(* IEC 61131-3 sources: ATCMcontrol_Engineering/src/COM/softing/fc/AddOns/Softing/4CPCTarget/Libs/ATCM_IEC1131_3/table_37, 6 files *)

(* ---- tof.st ---- *)
(*[[
    UserURL= "ATCM:TOF.htm"
]]*)
FUNCTION_BLOCK TOF

VAR_INPUT   (* Inputs *)
    IN : BOOL := FALSE; (* Input        *)
    PT : TIME := T#0s;  (* Preset time  *)
END_VAR

VAR_OUTPUT  (* Outputs *)
    Q  : BOOL := FALSE; (* FALSE if ET >= PT *)
    ET : TIME := T#0s;  (* Elapsed time      *)
END_VAR

VAR NON_RETAIN
    StartTime : TIME;
    Trig : BOOL := FALSE;
END_VAR

IF PT > T#0s THEN
    IF IN THEN
        Q := TRUE;
        ET := T#0s;
        Trig := FALSE;
    ELSIF NOT Trig THEN
        Trig := TRUE;
        StartTime := getTimeSinceSystemBoot();
    ELSIF Q THEN
        ET := getTimeSinceSystemBoot() - StartTime;
        IF ET >= PT THEN
            Q := FALSE;
            ET := PT;
        END_IF;
    END_IF;
ELSE
	(* error handling *)
    Q := IN;
    ET := T#0s;
    Trig := FALSE;
END_IF;

END_FUNCTION_BLOCK

(* ---- tof_ex.st ---- *)
(*[[
    UserURL= "ATCM:TOF_EX.htm"
]]*)
FUNCTION_BLOCK TOF_EX

VAR_INPUT   (* Inputs *)
    IN : BOOL := FALSE; (* Input        *)
    PT : TIME := T#0s;  (* Preset time  *)
END_VAR

VAR_INPUT (* Parameters *)
    SCALEMIN : DINT := 0;   (* minimum of scaling *)
    SCALEMAX : DINT := 100; (* maximum of scaling *)
END_VAR

VAR_OUTPUT  (* Outputs *)
    Q  : BOOL := FALSE; (* FALSE if ET >= PT *)
    ET : TIME := T#0s;  (* Elapsed time      *)
    ERROR : DINT;       (* Error             *)
END_VAR

VAR NON_RETAIN
    StartTime : TIME;
    Trig : BOOL := FALSE;
END_VAR

  ERROR := 0;
  IF (SCALEMIN >= SCALEMAX) THEN
     ERROR := -1;
  END_IF;

  IF PT > T#0s THEN
    IF IN THEN
        Q := TRUE;
        ET := T#0s;
        Trig := FALSE;
    ELSIF NOT Trig THEN
        Trig := TRUE;
        StartTime := getTimeSinceSystemBoot();
    ELSIF Q THEN
        ET := getTimeSinceSystemBoot() - StartTime;
        IF ET >= PT THEN
            Q := FALSE;
            ET := PT;
        END_IF;
    END_IF;
  ELSE
    (* error handling *)
    Q := IN;
    ET := T#0s;
    Trig := FALSE;
    ERROR := -1;
  END_IF;

END_FUNCTION_BLOCK

(* ---- ton.st ---- *)
(*[[
    UserURL= "ATCM:TON.htm"
]]*)
FUNCTION_BLOCK TON

VAR_INPUT   (* Inputs *)
    IN : BOOL := FALSE; (* Input        *)
    PT : TIME := T#0s;  (* Preset time 	*)
END_VAR

VAR_OUTPUT  (* Outputs *)
    Q  : BOOL := FALSE; (* TRUE if ET >= PT *)
    ET : TIME := T#0s;  (* Elapsed time     *)
END_VAR

VAR NON_RETAIN
    StartTime : TIME;
    Trig : BOOL := FALSE;
END_VAR

IF PT > T#0s THEN
    IF NOT IN THEN
        Q := FALSE;
        ET := T#0s;
		Trig := FALSE;
    ELSIF NOT Trig THEN
        Trig := TRUE;
        StartTime := getTimeSinceSystemBoot();
    ELSIF NOT Q THEN
        ET := getTimeSinceSystemBoot() - StartTime;
        IF ET >= PT THEN
            Q := TRUE;
            ET := PT;
        END_IF;
    END_IF;
ELSE
	(* error handling *)
    Q := IN;
    ET := T#0s;
    Trig := FALSE;
END_IF;

END_FUNCTION_BLOCK

(* ---- ton_ex.st ---- *)
(*[[
    UserURL= "ATCM:TON_EX.htm"
]]*)
FUNCTION_BLOCK TON_EX

VAR_INPUT   (* Inputs *)
    IN : BOOL := FALSE; (* Input        *)
    PT : TIME := T#0s;  (* Preset time 	*)
END_VAR

VAR_INPUT   (* Parameters *)
    SCALEMIN : DINT := 0;   (* minimum of scaling *)
    SCALEMAX : DINT := 100; (* maximum of scaling *)
END_VAR

VAR_OUTPUT  (* Outputs *)
    Q  : BOOL := FALSE; (* TRUE if ET >= PT *)
    ET : TIME := T#0s;  (* Elapsed time     *)
    ERROR : DINT;       (* error            *)
END_VAR

VAR NON_RETAIN
    StartTime : TIME;
    Trig : BOOL := FALSE;
END_VAR

  ERROR := 0;
  IF (SCALEMIN >= SCALEMAX) THEN
     ERROR := -1;
  END_IF;

  IF PT > T#0s THEN
    IF NOT IN THEN
        Q := FALSE;
        ET := T#0s;
        Trig := FALSE;
    ELSIF NOT Trig THEN
        Trig := TRUE;
        StartTime := getTimeSinceSystemBoot();
    ELSIF NOT Q THEN
        ET := getTimeSinceSystemBoot() - StartTime;
        IF ET >= PT THEN
            Q := TRUE;
            ET := PT;
        END_IF;
    END_IF;
  ELSE
    (* error handling *)
    Q := IN;
    ET := T#0s;
    Trig := FALSE;
    ERROR := -1;
  END_IF;

END_FUNCTION_BLOCK

(* ---- tp.st ---- *)
(*[[
    UserURL= "ATCM:TP.htm"
]]*)
FUNCTION_BLOCK TP

VAR_INPUT   (* Inputs *)
    IN : BOOL := FALSE; (* Input       *)
    PT : TIME := T#0s;  (* Preset time *)
END_VAR

VAR_OUTPUT  (* Outputs *)
    Q  : BOOL := FALSE; (* FALSE if ET >= PT    *)
    ET : TIME := T#0s;  (* Elapsed time         *)
END_VAR

VAR
    M         : BOOL := FALSE;
END_VAR

VAR NON_RETAIN
    Trig      : BOOL := FALSE;
    StartTime : TIME;
END_VAR

IF PT > T#0s THEN
    IF NOT Trig THEN
        Q := FALSE;
        IF IN AND NOT M THEN
            (* initilize function block *)
            (* get start time *)
            Trig := TRUE;
            StartTime := getTimeSinceSystemBoot();
            ET := T#0s;
            Q := TRUE;
        ELSIF NOT IN THEN
            ET := T#0s;
        END_IF;
    ELSE (* IF Trig *)
        (* get elapsed time *)
        ET := getTimeSinceSystemBoot() - Starttime;

        IF ET >= PT THEN (* time reached *)
            Trig := FALSE;
            Q := FALSE;
            IF NOT IN THEN
              ET := T#0s;
            ELSE
              ET := PT;
            END_IF;
        END_IF;
	END_IF;

ELSE
    (* error handling *)
    Q := FALSE;
    ET := T#0s;
    Trig := FALSE;
END_IF;

M := IN;

END_FUNCTION_BLOCK

(* ---- tp_ex.st ---- *)
(*[[
    UserURL= "ATCM:TP_EX.htm"
]]*)
FUNCTION_BLOCK TP_EX

VAR_INPUT   (* Inputs *)
    IN : BOOL := FALSE; (* Input       *)
    PT : TIME := T#0s;  (* Preset time *)
END_VAR

VAR_INPUT (* Parameters *)
    SCALEMIN : DINT := 0;   (* minimum of scaling *)
    SCALEMAX : DINT := 100; (* maximum of scaling *)
END_VAR

VAR_OUTPUT  (* Outputs *)
    Q  : BOOL := FALSE; (* FALSE if ET >= PT    *)
    ET : TIME := T#0s;  (* Elapsed time         *)
    ERROR : DINT;       (* Error                *)
END_VAR

VAR
    M         : BOOL := FALSE;
END_VAR

VAR NON_RETAIN
    Trig      : BOOL := FALSE;
    StartTime : TIME;
END_VAR

  ERROR := 0;
  IF (SCALEMIN >= SCALEMAX) THEN
     ERROR := -1;
  END_IF;

  IF PT > T#0s THEN
    IF NOT Trig THEN
        Q := FALSE;
        IF IN AND NOT M THEN
            (* initilize function block *)
            (* get start time *)
            Trig := TRUE;
            StartTime := getTimeSinceSystemBoot();
            ET := T#0s;
            Q := TRUE;
        ELSIF NOT IN THEN
            ET := T#0s;
        END_IF;
    ELSE (* IF Trig *)
        (* get elapsed time *)
        ET := getTimeSinceSystemBoot() - Starttime;

        IF ET >= PT THEN (* time reached *)
            Trig := FALSE;
            Q := FALSE;
            IF NOT IN THEN
              ET := T#0s;
            ELSE
              ET := PT;
            END_IF;
        END_IF;
	END_IF;

  ELSE
    (* error handling *)
    Q := FALSE;
    ET := T#0s;
    Trig := FALSE;
    ERROR := -1;
  END_IF;

  M := IN;

END_FUNCTION_BLOCK
